# EPICS IOC start-up script: iocs/exampleIOC/iocBoot/iocExample/settings.iocsh
# prefix used for all PVs in this IOC
epicsEnvSet("PREFIX", "example:")
